TYPE ST_DS_Zustand :
STRUCT
	Druck	: REAL;

	Warnung				: BOOL;
	Warnung_Code		: WORD;
END_STRUCT
END_TYPE

(* stored: Version 1.1.0.1, ProductVersion 3.1.4024.9
   DUT ST_DS_Zustand: Id {a8844baf-e7fb-4c09-8275-46badcde27ad} *)
